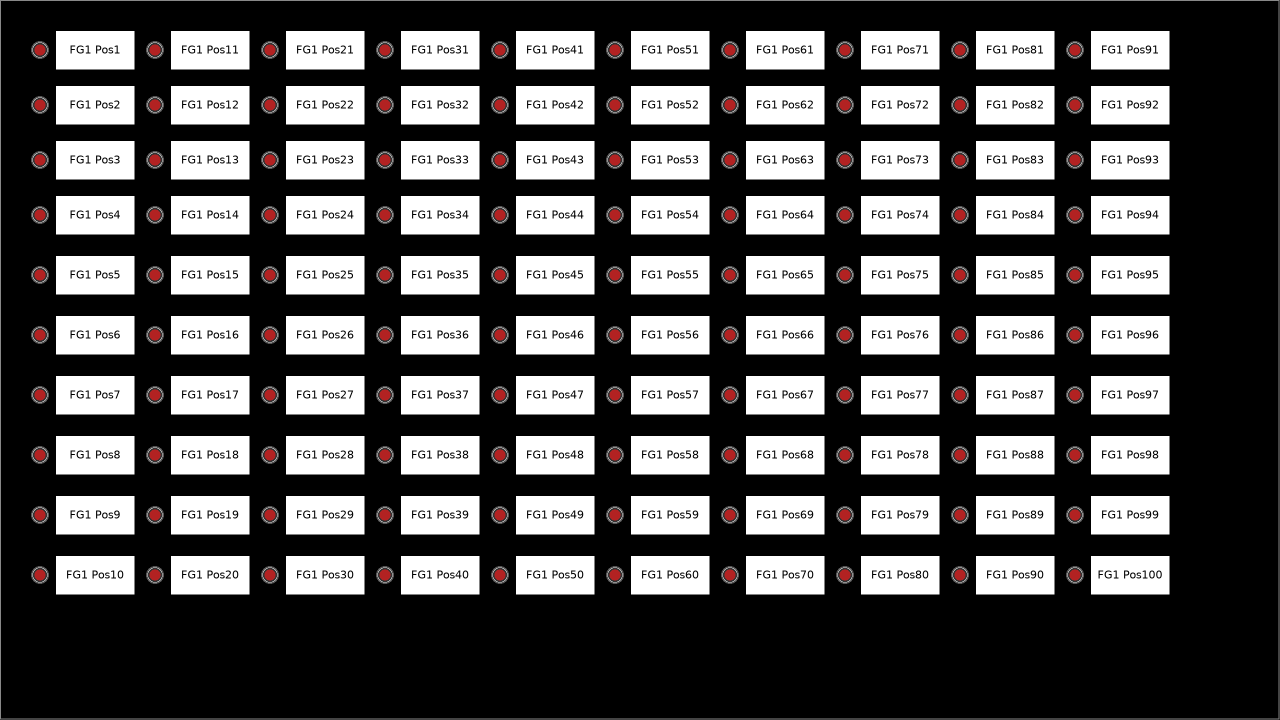
VISUALIZATION PAGE_KR1_Tab_1_100  // 1280x720
    RoundedRectangle (170,30 80x40), "FG1 Pos11"
        toggle KR1.bOutBit[5,4]
        OnMouseClick: execute {  }
    Lamp1 (145,40 20x20), variable: KR1.bInBit[5,4], style: Lamp-Lamp1-Red
    RoundedRectangle (55,30 80x40), "FG1 Pos1"
        toggle KR1.bOutBit[4,2]
        OnMouseClick: execute {  }
    Lamp1 (30,40 20x20), variable: KR1.bInBit[4,2], style: Lamp-Lamp1-Red
    RoundedRectangle (285,30 80x40), "FG1 Pos21"
        toggle KR1.bOutBit[6,6]
        OnMouseClick: execute {  }
    Lamp1 (260,40 20x20), variable: KR1.bInBit[6,6], style: Lamp-Lamp1-Red
    RoundedRectangle (400,30 80x40), "FG1 Pos31"
        toggle KR1.bOutBit[8,0]
        OnMouseClick: execute {  }
    Lamp1 (375,40 20x20), variable: KR1.bInBit[8,0], style: Lamp-Lamp1-Red
    RoundedRectangle (515,30 80x40), "FG1 Pos41"
        toggle KR1.bOutBit[9,2]
        OnMouseClick: execute {  }
    Lamp1 (490,40 20x20), variable: KR1.bInBit[9,2], style: Lamp-Lamp1-Red
    RoundedRectangle (745,30 80x40), "FG1 Pos61"
        toggle KR1.bOutBit[11,6]
        OnMouseClick: execute {  }
    Lamp1 (720,40 20x20), variable: KR1.bInBit[11,6], style: Lamp-Lamp1-Red
    RoundedRectangle (630,30 80x40), "FG1 Pos51"
        toggle KR1.bOutBit[10,4]
        OnMouseClick: execute {  }
    Lamp1 (605,40 20x20), variable: KR1.bInBit[10,4], style: Lamp-Lamp1-Red
    RoundedRectangle (860,30 80x40), "FG1 Pos71"
        toggle KR1.bOutBit[13,0]
        OnMouseClick: execute {  }
    Lamp1 (835,40 20x20), variable: KR1.bInBit[13,0], style: Lamp-Lamp1-Red
    RoundedRectangle (975,30 80x40), "FG1 Pos81"
        toggle KR1.bOutBit[14,2]
        OnMouseClick: execute {  }
    Lamp1 (950,40 20x20), variable: KR1.bInBit[14,2], style: Lamp-Lamp1-Red
    RoundedRectangle (1090,30 80x40), "FG1 Pos91"
        toggle KR1.bOutBit[15,4]
        OnMouseClick: execute {  }
    Lamp1 (1065,40 20x20), variable: KR1.bInBit[15,4], style: Lamp-Lamp1-Red
    RoundedRectangle (170,85 80x40), "FG1 Pos12"
        toggle KR1.bOutBit[5,5]
        OnMouseClick: execute {  }
    Lamp1 (145,95 20x20), variable: KR1.bInBit[5,5], style: Lamp-Lamp1-Red
    RoundedRectangle (55,85 80x40), "FG1 Pos2"
        toggle KR1.bOutBit[4,3]
        OnMouseClick: execute {  }
    Lamp1 (30,95 20x20), variable: KR1.bInBit[4,3], style: Lamp-Lamp1-Red
    RoundedRectangle (285,85 80x40), "FG1 Pos22"
        toggle KR1.bOutBit[6,7]
        OnMouseClick: execute {  }
    Lamp1 (260,95 20x20), variable: KR1.bInBit[6,7], style: Lamp-Lamp1-Red
    RoundedRectangle (400,85 80x40), "FG1 Pos32"
        toggle KR1.bOutBit[8,1]
        OnMouseClick: execute {  }
    Lamp1 (375,95 20x20), variable: KR1.bInBit[8,1], style: Lamp-Lamp1-Red
    RoundedRectangle (515,85 80x40), "FG1 Pos42"
        toggle KR1.bOutBit[9,3]
        OnMouseClick: execute {  }
    Lamp1 (490,95 20x20), variable: KR1.bInBit[9,3], style: Lamp-Lamp1-Red
    RoundedRectangle (745,85 80x40), "FG1 Pos62"
        toggle KR1.bOutBit[11,7]
        OnMouseClick: execute {  }
    Lamp1 (720,95 20x20), variable: KR1.bInBit[11,7], style: Lamp-Lamp1-Red
    RoundedRectangle (630,85 80x40), "FG1 Pos52"
        toggle KR1.bOutBit[10,5]
        OnMouseClick: execute {  }
    Lamp1 (605,95 20x20), variable: KR1.bInBit[10,5], style: Lamp-Lamp1-Red
    RoundedRectangle (860,85 80x40), "FG1 Pos72"
        toggle KR1.bOutBit[13,1]
        OnMouseClick: execute {  }
    Lamp1 (835,95 20x20), variable: KR1.bInBit[13,1], style: Lamp-Lamp1-Red
    RoundedRectangle (975,85 80x40), "FG1 Pos82"
        toggle KR1.bOutBit[14,3]
        OnMouseClick: execute {  }
    Lamp1 (950,95 20x20), variable: KR1.bInBit[14,3], style: Lamp-Lamp1-Red
    RoundedRectangle (1090,85 80x40), "FG1 Pos92"
        toggle KR1.bOutBit[15,5]
        OnMouseClick: execute {  }
    Lamp1 (1065,95 20x20), variable: KR1.bInBit[15,5], style: Lamp-Lamp1-Red
    RoundedRectangle (170,140 80x40), "FG1 Pos13"
        toggle KR1.bOutBit[5,6]
        OnMouseClick: execute {  }
    Lamp1 (145,150 20x20), variable: KR1.bInBit[5,6], style: Lamp-Lamp1-Red
    RoundedRectangle (55,140 80x40), "FG1 Pos3"
        toggle KR1.bOutBit[4,4]
        OnMouseClick: execute {  }
    Lamp1 (30,150 20x20), variable: KR1.bInBit[4,4], style: Lamp-Lamp1-Red
    RoundedRectangle (285,140 80x40), "FG1 Pos23"
        toggle KR1.bOutBit[7,0]
        OnMouseClick: execute {  }
    Lamp1 (260,150 20x20), variable: KR1.bInBit[7,0], style: Lamp-Lamp1-Red
    RoundedRectangle (400,140 80x40), "FG1 Pos33"
        toggle KR1.bOutBit[8,2]
        OnMouseClick: execute {  }
    Lamp1 (375,150 20x20), variable: KR1.bInBit[8,2], style: Lamp-Lamp1-Red
    RoundedRectangle (515,140 80x40), "FG1 Pos43"
        toggle KR1.bOutBit[9,4]
        OnMouseClick: execute {  }
    Lamp1 (490,150 20x20), variable: KR1.bInBit[9,4], style: Lamp-Lamp1-Red
    RoundedRectangle (745,140 80x40), "FG1 Pos63"
        toggle KR1.bOutBit[12,0]
        OnMouseClick: execute {  }
    Lamp1 (720,150 20x20), variable: KR1.bInBit[12,0], style: Lamp-Lamp1-Red
    RoundedRectangle (630,140 80x40), "FG1 Pos53"
        toggle KR1.bOutBit[10,6]
        OnMouseClick: execute {  }
    Lamp1 (605,150 20x20), variable: KR1.bInBit[10,6], style: Lamp-Lamp1-Red
    RoundedRectangle (860,140 80x40), "FG1 Pos73"
        toggle KR1.bOutBit[13,2]
        OnMouseClick: execute {  }
    Lamp1 (835,150 20x20), variable: KR1.bInBit[13,2], style: Lamp-Lamp1-Red
    RoundedRectangle (975,140 80x40), "FG1 Pos83"
        toggle KR1.bOutBit[14,4]
        OnMouseClick: execute {  }
    Lamp1 (950,150 20x20), variable: KR1.bInBit[14,4], style: Lamp-Lamp1-Red
    RoundedRectangle (1090,140 80x40), "FG1 Pos93"
        toggle KR1.bOutBit[15,6]
        OnMouseClick: execute {  }
    Lamp1 (1065,150 20x20), variable: KR1.bInBit[15,6], style: Lamp-Lamp1-Red
    RoundedRectangle (170,195 80x40), "FG1 Pos14"
        toggle KR1.bOutBit[5,7]
        OnMouseClick: execute {  }
    Lamp1 (145,205 20x20), variable: KR1.bInBit[5,7], style: Lamp-Lamp1-Red
    RoundedRectangle (55,195 80x40), "FG1 Pos4"
        toggle KR1.bOutBit[4,5]
        OnMouseClick: execute {  }
    Lamp1 (30,205 20x20), variable: KR1.bInBit[4,5], style: Lamp-Lamp1-Red
    RoundedRectangle (285,195 80x40), "FG1 Pos24"
        toggle KR1.bOutBit[7,1]
        OnMouseClick: execute {  }
    Lamp1 (260,205 20x20), variable: KR1.bInBit[7,1], style: Lamp-Lamp1-Red
    RoundedRectangle (400,195 80x40), "FG1 Pos34"
        toggle KR1.bOutBit[8,3]
        OnMouseClick: execute {  }
    Lamp1 (375,205 20x20), variable: KR1.bInBit[8,3], style: Lamp-Lamp1-Red
    RoundedRectangle (515,195 80x40), "FG1 Pos44"
        toggle KR1.bOutBit[9,5]
        OnMouseClick: execute {  }
    Lamp1 (490,205 20x20), variable: KR1.bInBit[9,5], style: Lamp-Lamp1-Red
    RoundedRectangle (745,195 80x40), "FG1 Pos64"
        toggle KR1.bOutBit[12,1]
        OnMouseClick: execute {  }
    Lamp1 (720,205 20x20), variable: KR1.bInBit[12,1], style: Lamp-Lamp1-Red
    RoundedRectangle (630,195 80x40), "FG1 Pos54"
        toggle KR1.bOutBit[10,7]
        OnMouseClick: execute {  }
    Lamp1 (605,205 20x20), variable: KR1.bInBit[10,7], style: Lamp-Lamp1-Red
    RoundedRectangle (860,195 80x40), "FG1 Pos74"
        toggle KR1.bOutBit[13,3]
        OnMouseClick: execute {  }
    Lamp1 (835,205 20x20), variable: KR1.bInBit[13,3], style: Lamp-Lamp1-Red
    RoundedRectangle (975,195 80x40), "FG1 Pos84"
        toggle KR1.bOutBit[14,5]
        OnMouseClick: execute {  }
    Lamp1 (950,205 20x20), variable: KR1.bInBit[14,5], style: Lamp-Lamp1-Red
    RoundedRectangle (1090,195 80x40), "FG1 Pos94"
        toggle KR1.bOutBit[15,7]
        OnMouseClick: execute {  }
    Lamp1 (1065,205 20x20), variable: KR1.bInBit[15,7], style: Lamp-Lamp1-Red
    RoundedRectangle (170,255 80x40), "FG1 Pos15"
        toggle KR1.bOutBit[6,0]
        OnMouseClick: execute {  }
    Lamp1 (145,265 20x20), variable: KR1.bInBit[6,0], style: Lamp-Lamp1-Red
    RoundedRectangle (55,255 80x40), "FG1 Pos5"
        toggle KR1.bOutBit[4,6]
        OnMouseClick: execute {  }
    Lamp1 (30,265 20x20), variable: KR1.bInBit[4,6], style: Lamp-Lamp1-Red
    RoundedRectangle (285,255 80x40), "FG1 Pos25"
        toggle KR1.bOutBit[7,2]
        OnMouseClick: execute {  }
    Lamp1 (260,265 20x20), variable: KR1.bInBit[7,2], style: Lamp-Lamp1-Red
    RoundedRectangle (400,255 80x40), "FG1 Pos35"
        toggle KR1.bOutBit[8,4]
        OnMouseClick: execute {  }
    Lamp1 (375,265 20x20), variable: KR1.bInBit[8,4], style: Lamp-Lamp1-Red
    RoundedRectangle (515,255 80x40), "FG1 Pos45"
        toggle KR1.bOutBit[9,6]
        OnMouseClick: execute {  }
    Lamp1 (490,265 20x20), variable: KR1.bInBit[9,6], style: Lamp-Lamp1-Red
    RoundedRectangle (745,255 80x40), "FG1 Pos65"
        toggle KR1.bOutBit[12,2]
        OnMouseClick: execute {  }
    Lamp1 (720,265 20x20), variable: KR1.bInBit[12,2], style: Lamp-Lamp1-Red
    RoundedRectangle (630,255 80x40), "FG1 Pos55"
        toggle KR1.bOutBit[11,0]
        OnMouseClick: execute {  }
    Lamp1 (605,265 20x20), variable: KR1.bInBit[11,0], style: Lamp-Lamp1-Red
    RoundedRectangle (860,255 80x40), "FG1 Pos75"
        toggle KR1.bOutBit[13,4]
        OnMouseClick: execute {  }
    Lamp1 (835,265 20x20), variable: KR1.bInBit[13,4], style: Lamp-Lamp1-Red
    RoundedRectangle (975,255 80x40), "FG1 Pos85"
        toggle KR1.bOutBit[14,6]
        OnMouseClick: execute {  }
    Lamp1 (950,265 20x20), variable: KR1.bInBit[14,6], style: Lamp-Lamp1-Red
    RoundedRectangle (1090,255 80x40), "FG1 Pos95"
        toggle KR1.bOutBit[16,0]
        OnMouseClick: execute {  }
    Lamp1 (1065,265 20x20), variable: KR1.bInBit[16,0], style: Lamp-Lamp1-Red
    RoundedRectangle (170,315 80x40), "FG1 Pos16"
        toggle KR1.bOutBit[6,1]
        OnMouseClick: execute {  }
    Lamp1 (145,325 20x20), variable: KR1.bInBit[6,1], style: Lamp-Lamp1-Red
    RoundedRectangle (55,315 80x40), "FG1 Pos6"
        toggle KR1.bOutBit[4,7]
        OnMouseClick: execute {  }
    Lamp1 (30,325 20x20), variable: KR1.bInBit[4,7], style: Lamp-Lamp1-Red
    RoundedRectangle (285,315 80x40), "FG1 Pos26"
        toggle KR1.bOutBit[7,3]
        OnMouseClick: execute {  }
    Lamp1 (260,325 20x20), variable: KR1.bInBit[7,3], style: Lamp-Lamp1-Red
    RoundedRectangle (400,315 80x40), "FG1 Pos36"
        toggle KR1.bOutBit[8,5]
        OnMouseClick: execute {  }
    Lamp1 (375,325 20x20), variable: KR1.bInBit[8,5], style: Lamp-Lamp1-Red
    RoundedRectangle (515,315 80x40), "FG1 Pos46"
        toggle KR1.bOutBit[9,7]
        OnMouseClick: execute {  }
    Lamp1 (490,325 20x20), variable: KR1.bInBit[9,7], style: Lamp-Lamp1-Red
    RoundedRectangle (745,315 80x40), "FG1 Pos66"
        toggle KR1.bOutBit[12,3]
        OnMouseClick: execute {  }
    Lamp1 (720,325 20x20), variable: KR1.bInBit[12,3], style: Lamp-Lamp1-Red
    RoundedRectangle (630,315 80x40), "FG1 Pos56"
        toggle KR1.bOutBit[11,1]
        OnMouseClick: execute {  }
    Lamp1 (605,325 20x20), variable: KR1.bInBit[11,1], style: Lamp-Lamp1-Red
    RoundedRectangle (860,315 80x40), "FG1 Pos76"
        toggle KR1.bOutBit[13,5]
        OnMouseClick: execute {  }
    Lamp1 (835,325 20x20), variable: KR1.bInBit[13,5], style: Lamp-Lamp1-Red
    RoundedRectangle (975,315 80x40), "FG1 Pos86"
        toggle KR1.bOutBit[14,7]
        OnMouseClick: execute {  }
    Lamp1 (950,325 20x20), variable: KR1.bInBit[14,7], style: Lamp-Lamp1-Red
    RoundedRectangle (1090,315 80x40), "FG1 Pos96"
        toggle KR1.bOutBit[16,1]
        OnMouseClick: execute {  }
    Lamp1 (1065,325 20x20), variable: KR1.bInBit[16,1], style: Lamp-Lamp1-Red
    RoundedRectangle (170,375 80x40), "FG1 Pos17"
        toggle KR1.bOutBit[6,2]
        OnMouseClick: execute {  }
    Lamp1 (145,385 20x20), variable: KR1.bInBit[6,2], style: Lamp-Lamp1-Red
    RoundedRectangle (55,375 80x40), "FG1 Pos7"
        toggle KR1.bOutBit[5,0]
        OnMouseClick: execute {  }
    Lamp1 (30,385 20x20), variable: KR1.bInBit[5,0], style: Lamp-Lamp1-Red
    RoundedRectangle (285,375 80x40), "FG1 Pos27"
        toggle KR1.bOutBit[7,4]
        OnMouseClick: execute {  }
    Lamp1 (260,385 20x20), variable: KR1.bInBit[7,4], style: Lamp-Lamp1-Red
    RoundedRectangle (400,375 80x40), "FG1 Pos37"
        toggle KR1.bOutBit[8,6]
        OnMouseClick: execute {  }
    Lamp1 (375,385 20x20), variable: KR1.bInBit[8,6], style: Lamp-Lamp1-Red
    RoundedRectangle (515,375 80x40), "FG1 Pos47"
        toggle KR1.bOutBit[10,0]
        OnMouseClick: execute {  }
    Lamp1 (490,385 20x20), variable: KR1.bInBit[10,0], style: Lamp-Lamp1-Red
    RoundedRectangle (745,375 80x40), "FG1 Pos67"
        toggle KR1.bOutBit[12,4]
        OnMouseClick: execute {  }
    Lamp1 (720,385 20x20), variable: KR1.bInBit[12,4], style: Lamp-Lamp1-Red
    RoundedRectangle (630,375 80x40), "FG1 Pos57"
        toggle KR1.bOutBit[11,2]
        OnMouseClick: execute {  }
    Lamp1 (605,385 20x20), variable: KR1.bInBit[11,2], style: Lamp-Lamp1-Red
    RoundedRectangle (860,375 80x40), "FG1 Pos77"
        toggle KR1.bOutBit[13,6]
        OnMouseClick: execute {  }
    Lamp1 (835,385 20x20), variable: KR1.bInBit[13,6], style: Lamp-Lamp1-Red
    RoundedRectangle (975,375 80x40), "FG1 Pos87"
        toggle KR1.bOutBit[15,0]
        OnMouseClick: execute {  }
    Lamp1 (950,385 20x20), variable: KR1.bInBit[15,0], style: Lamp-Lamp1-Red
    RoundedRectangle (1090,375 80x40), "FG1 Pos97"
        toggle KR1.bOutBit[16,2]
        OnMouseClick: execute {  }
    Lamp1 (1065,385 20x20), variable: KR1.bInBit[16,2], style: Lamp-Lamp1-Red
    RoundedRectangle (170,435 80x40), "FG1 Pos18"
        toggle KR1.bOutBit[6,3]
        OnMouseClick: execute {  }
    Lamp1 (145,445 20x20), variable: KR1.bInBit[6,3], style: Lamp-Lamp1-Red
    RoundedRectangle (55,435 80x40), "FG1 Pos8"
        toggle KR1.bOutBit[5,1]
        OnMouseClick: execute {  }
    Lamp1 (30,445 20x20), variable: KR1.bInBit[5,1], style: Lamp-Lamp1-Red
    RoundedRectangle (285,435 80x40), "FG1 Pos28"
        toggle KR1.bOutBit[7,5]
        OnMouseClick: execute {  }
    Lamp1 (260,445 20x20), variable: KR1.bInBit[7,5], style: Lamp-Lamp1-Red
    RoundedRectangle (400,435 80x40), "FG1 Pos38"
        toggle KR1.bOutBit[8,7]
        OnMouseClick: execute {  }
    Lamp1 (375,445 20x20), variable: KR1.bInBit[8,7], style: Lamp-Lamp1-Red
    RoundedRectangle (515,435 80x40), "FG1 Pos48"
        toggle KR1.bOutBit[10,1]
        OnMouseClick: execute {  }
    Lamp1 (490,445 20x20), variable: KR1.bInBit[10,1], style: Lamp-Lamp1-Red
    RoundedRectangle (745,435 80x40), "FG1 Pos68"
        toggle KR1.bOutBit[12,5]
        OnMouseClick: execute {  }
    Lamp1 (720,445 20x20), variable: KR1.bInBit[12,5], style: Lamp-Lamp1-Red
    RoundedRectangle (630,435 80x40), "FG1 Pos58"
        toggle KR1.bOutBit[11,3]
        OnMouseClick: execute {  }
    Lamp1 (605,445 20x20), variable: KR1.bInBit[11,3], style: Lamp-Lamp1-Red
    RoundedRectangle (860,435 80x40), "FG1 Pos78"
        toggle KR1.bOutBit[13,7]
        OnMouseClick: execute {  }
    Lamp1 (835,445 20x20), variable: KR1.bInBit[13,7], style: Lamp-Lamp1-Red
    RoundedRectangle (975,435 80x40), "FG1 Pos88"
        toggle KR1.bOutBit[15,1]
        OnMouseClick: execute {  }
    Lamp1 (950,445 20x20), variable: KR1.bInBit[15,1], style: Lamp-Lamp1-Red
    RoundedRectangle (1090,435 80x40), "FG1 Pos98"
        toggle KR1.bOutBit[16,3]
        OnMouseClick: execute {  }
    Lamp1 (1065,445 20x20), variable: KR1.bInBit[16,3], style: Lamp-Lamp1-Red
    RoundedRectangle (55,495 80x40), "FG1 Pos9"
        toggle KR1.bOutBit[5,2]
        OnMouseClick: execute {  }
    Lamp1 (30,505 20x20), variable: KR1.bInBit[5,2], style: Lamp-Lamp1-Red
    RoundedRectangle (170,495 80x40), "FG1 Pos19"
        toggle KR1.bOutBit[6,4]
        OnMouseClick: execute {  }
    Lamp1 (145,505 20x20), variable: KR1.bInBit[6,4], style: Lamp-Lamp1-Red
    RoundedRectangle (285,495 80x40), "FG1 Pos29"
        toggle KR1.bOutBit[7,6]
        OnMouseClick: execute {  }
    Lamp1 (260,505 20x20), variable: KR1.bInBit[7,6], style: Lamp-Lamp1-Red
    RoundedRectangle (400,495 80x40), "FG1 Pos39"
        toggle KR1.bOutBit[9,0]
        OnMouseClick: execute {  }
    Lamp1 (375,505 20x20), variable: KR1.bInBit[9,0], style: Lamp-Lamp1-Red
    RoundedRectangle (515,495 80x40), "FG1 Pos49"
        toggle KR1.bOutBit[10,2]
        OnMouseClick: execute {  }
    Lamp1 (490,505 20x20), variable: KR1.bInBit[10,2], style: Lamp-Lamp1-Red
    RoundedRectangle (630,495 80x40), "FG1 Pos59"
        toggle KR1.bOutBit[11,4]
        OnMouseClick: execute {  }
    Lamp1 (605,505 20x20), variable: KR1.bInBit[11,4], style: Lamp-Lamp1-Red
    RoundedRectangle (745,495 80x40), "FG1 Pos69"
        toggle KR1.bOutBit[12,6]
        OnMouseClick: execute {  }
    Lamp1 (720,505 20x20), variable: KR1.bInBit[12,6], style: Lamp-Lamp1-Red
    RoundedRectangle (860,495 80x40), "FG1 Pos79"
        toggle KR1.bOutBit[14,0]
        OnMouseClick: execute {  }
    Lamp1 (835,505 20x20), variable: KR1.bInBit[14,0], style: Lamp-Lamp1-Red
    RoundedRectangle (975,495 80x40), "FG1 Pos89"
        toggle KR1.bOutBit[15,2]
        OnMouseClick: execute {  }
    Lamp1 (950,505 20x20), variable: KR1.bInBit[15,2], style: Lamp-Lamp1-Red
    RoundedRectangle (1090,495 80x40), "FG1 Pos99"
        toggle KR1.bOutBit[16,4]
        OnMouseClick: execute {  }
    Lamp1 (1065,505 20x20), variable: KR1.bInBit[16,4], style: Lamp-Lamp1-Red
    RoundedRectangle (55,555 80x40), "FG1 Pos10"
        toggle KR1.bOutBit[5,3]
        OnMouseClick: execute {  }
    Lamp1 (30,565 20x20), variable: KR1.bInBit[5,3], style: Lamp-Lamp1-Red
    RoundedRectangle (170,555 80x40), "FG1 Pos20"
        toggle KR1.bOutBit[6,5]
        OnMouseClick: execute {  }
    Lamp1 (145,565 20x20), variable: KR1.bInBit[6,5], style: Lamp-Lamp1-Red
    RoundedRectangle (285,555 80x40), "FG1 Pos30"
        toggle KR1.bOutBit[7,7]
        OnMouseClick: execute {  }
    Lamp1 (260,565 20x20), variable: KR1.bInBit[7,7], style: Lamp-Lamp1-Red
    RoundedRectangle (400,555 80x40), "FG1 Pos40"
        toggle KR1.bOutBit[9,1]
        OnMouseClick: execute {  }
    Lamp1 (375,565 20x20), variable: KR1.bInBit[9,1], style: Lamp-Lamp1-Red
    RoundedRectangle (515,555 80x40), "FG1 Pos50"
        toggle KR1.bOutBit[10,3]
        OnMouseClick: execute {  }
    Lamp1 (490,565 20x20), variable: KR1.bInBit[10,3], style: Lamp-Lamp1-Red
    RoundedRectangle (630,555 80x40), "FG1 Pos60"
        toggle KR1.bOutBit[11,5]
        OnMouseClick: execute {  }
    Lamp1 (605,565 20x20), variable: KR1.bInBit[11,5], style: Lamp-Lamp1-Red
    RoundedRectangle (745,555 80x40), "FG1 Pos70"
        toggle KR1.bOutBit[12,7]
        OnMouseClick: execute {  }
    Lamp1 (720,565 20x20), variable: KR1.bInBit[12,7], style: Lamp-Lamp1-Red
    RoundedRectangle (860,555 80x40), "FG1 Pos80"
        toggle KR1.bOutBit[14,1]
        OnMouseClick: execute {  }
    Lamp1 (835,565 20x20), variable: KR1.bInBit[14,1], style: Lamp-Lamp1-Red
    RoundedRectangle (975,555 80x40), "FG1 Pos90"
        toggle KR1.bOutBit[15,3]
        OnMouseClick: execute {  }
    Lamp1 (950,565 20x20), variable: KR1.bInBit[15,3], style: Lamp-Lamp1-Red
    RoundedRectangle (1090,555 80x40), "FG1 Pos100"
        toggle KR1.bOutBit[16,5]
        OnMouseClick: execute {  }
    Lamp1 (1065,565 20x20), variable: KR1.bInBit[16,5], style: Lamp-Lamp1-Red
END_VISUALIZATION

(* stored: Version 1.1.0.1, ProductVersion 3.1.4024.12
   Visu PAGE_KR1_Tab_1_100: Id {b15b5380-33d3-43fd-8a5d-d43db15c6877} *)
